SUBAPPLICATION Uebung_004b3 (* Toggle Flip-Flop mit IE / Split / Verriegelt *)
  (* Standard: 61499-2; Description: Copyright (c) 2023 Meisterschulen am Ostbahnhof This program and the accompanying materials are made available under the terms of the Eclipse Public License 2.0 which is available at https://www.eclipse.org/legal/epl-2.0/ SPDX-License-Identifier: EPL-2.0 *)
  (* Version 1.0, 2023-10-23, Franz Höpfinger, Meisterschulen am Ostbahnhof, initial API and implementation and/or initial documentation *)
  PACKAGE Uebungen;
  IMPORT logiBUS::io::DI::logiBUS_DI::Input_I1;
  IMPORT logiBUS::io::DI::logiBUS_DI::Input_I2;
  IMPORT logiBUS::io::DI::logiBUS_DI_Events::BUTTON_SINGLE_CLICK;
  IMPORT logiBUS::io::DQ::logiBUS_DO::Output_Q1;
  IMPORT logiBUS::io::DQ::logiBUS_DO::Output_Q2;
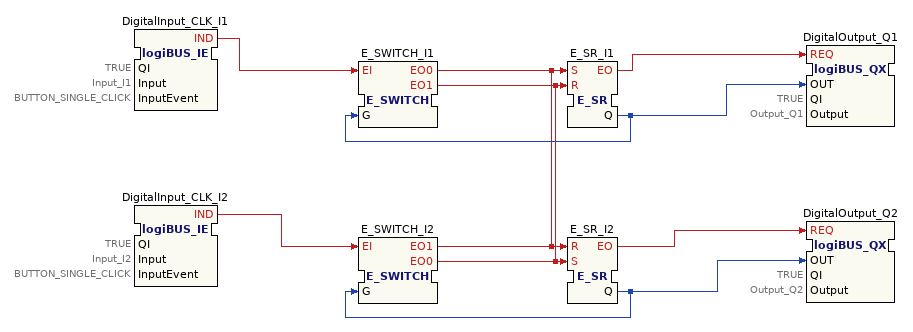
  FBS
    DigitalOutput_Q1 : logiBUS::io::DQ::logiBUS_QX(QI := TRUE, Output := Output_Q1);
    DigitalInput_CLK_I1 : logiBUS::io::DI::logiBUS_IE(QI := TRUE, Input := Input_I1, InputEvent := BUTTON_SINGLE_CLICK);
    E_SR_I1 : iec61499::events::E_SR;
    E_SWITCH_I1 : iec61499::events::E_SWITCH;
    E_SWITCH_I2 : iec61499::events::E_SWITCH;
    DigitalOutput_Q2 : logiBUS::io::DQ::logiBUS_QX(QI := TRUE, Output := Output_Q2);
    E_SR_I2 : iec61499::events::E_SR;
    DigitalInput_CLK_I2 : logiBUS::io::DI::logiBUS_IE(QI := TRUE, Input := Input_I2, InputEvent := BUTTON_SINGLE_CLICK);
  END_FBS
  EVENT_CONNECTIONS
    E_SR_I1.EO TO DigitalOutput_Q1.REQ;
    DigitalInput_CLK_I1.IND TO E_SWITCH_I1.EI;
    E_SWITCH_I1.EO0 TO E_SR_I1.S;
    E_SWITCH_I1.EO1 TO E_SR_I1.R;
    E_SWITCH_I2.EO1 TO E_SR_I2.R;
    E_SWITCH_I2.EO0 TO E_SR_I2.S;
    E_SR_I2.EO TO DigitalOutput_Q2.REQ;
    DigitalInput_CLK_I2.IND TO E_SWITCH_I2.EI;
    E_SWITCH_I2.EO0 TO E_SR_I1.R;
    E_SWITCH_I1.EO0 TO E_SR_I2.R;
  END_CONNECTIONS
  DATA_CONNECTIONS
    E_SR_I1.Q TO DigitalOutput_Q1.OUT;
    E_SR_I1.Q TO E_SWITCH_I1.G;
    E_SR_I2.Q TO E_SWITCH_I2.G;
    E_SR_I2.Q TO DigitalOutput_Q2.OUT;
  END_CONNECTIONS
END_SUBAPPLICATION
